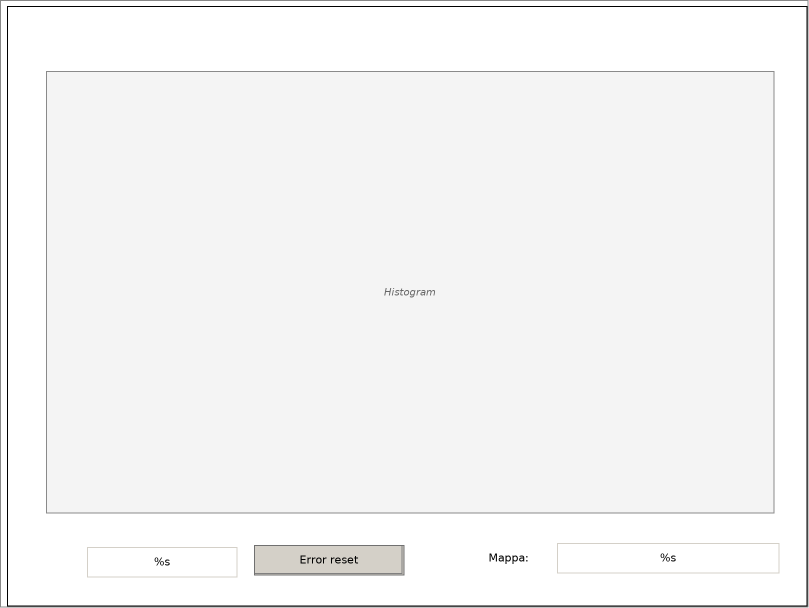
VISUALIZATION HegesztesGrafikon  // 809x608
    Rectangle (7,6 800x600)
    Histogram (46,71 728x442), scale format: %.1f, scale 0..3000
        p1518820177: HEGESZTESUTMERES.nDistances
        p102497268: HEGESZTESUTMERES.nDistances
        p788070771: ARRAY [0..3000] OF DINT
    Button (254,545 150x30), "Error reset"
        OnMouseClick: execute { HEGESZTESUTMERES.iState:=1; }
    Textfield (87,547 150x30), "%s", text variable: HEGESZTESUTMERES.iState, colour toggle: HEGESZTESUTMERES.bError, colour variable: HEGESZTESUTMERES.nNormalFillColor
        p2167032090: HEGESZTESUTMERES.nAlarmFillColor
    Textfield (557,543 222x30), "%s", text variable: HEGESZTESUTMERES.sFolder
        OnMouseClick: write HEGESZTESUTMERES.sFolder via VisuDialogs.Keypad
    Label (470,543 77x30), "Mappa:"
END_VISUALIZATION

(* stored: Version 1.1.0.1, ProductVersion 3.1.4024.11
   Visu HegesztesGrafikon: Id {b05781ff-62a1-4296-a20a-affda320981a} *)
